FUNCTION_BLOCK "G269M_Code"
TITLE =G269M TEMPERATURE MES. KILN 1
//COPYRIGHT:    (C) 2009  BUHLER AG, CH-9240 UZWIL, SWITZERLAND
//
//PRODUCT:      WinCoS_BIW01_09
//
//TITLE:        TEMPERATURE MES. KILN 1
//                Machine group control
//                Maschinengruppensteuerung
//
//--------------------------------------------------------------------------------
//
//IDENT:        AUTHOR:             DEPT:                              DATE:
//
//P01_FB369.1.0 K.Renz              CSB41                              30.Sep.2009
//             1st Release
//
//--------------------------------------------------------------------------------
//
//PURPOSE:
//
//MANUAL :
//
//RESTRICTIONS:
//
//--------------------------------------------------------------------------------
AUTHOR : KR
FAMILY : USW
VERSION : 9.9


VAR
  Gr : "GCS7_GrpCtrlSub";	//Standard interface to group
  InOutValue1 : DINT ;	//Data for user
  InOutValue2 : DINT ;	//Data for user
  OutWayConflict : BOOL ;	//Data for user
  OutSelectionOk : BOOL ;	//Data for user
  CmdNewValue : BOOL ;	//Data for user
  CmdNewJob : BOOL ;	//Data for user
  OutCodeOK : BOOL ;	//Data for user
  InEndOfJob : BOOL ;	//Data for user
  staWayOk : BOOL ;	//Data for user
  EdgeStartRelease : BOOL ;	//Data for user
  read_3191 : BOOL ;	//Data for user
  USW9 : BOOL ;	//Data for user
  USW10 : BOOL ;	//Data for user
  USW11 : BOOL ;	//Data for user
  USW12 : BOOL ;	//Data for user
  USW13 : BOOL ;	//Data for user
  USW14 : BOOL ;	//Data for user
  USW15 : BOOL ;	//Data for user
  A_3191_BTE01 : "GCS7_E_AnalogInput";	// AnaInp
  A_3191_BTE05 : "GCS7_E_AnalogInput";	// AnaInp
  A_3191_BTE07 : "GCS7_E_AnalogInput";	// AnaInp
  A_3191_BTE08 : "GCS7_E_AnalogInput";	// AnaInp
  A_3191_BTE10 : "GCS7_E_AnalogInput";	// AnaInp
  A_3191_BTE11 : "GCS7_E_AnalogInput";	// AnaInp
  A_3191_BTE12 : "GCS7_E_AnalogInput";	// AnaInp
  A_3191_BTE06 : "GCS7_E_AnalogInput";	// AnaInp
  A_3191_BTE13 : "GCS7_E_AnalogInput";	// AnaInp
END_VAR
VAR_TEMP
  tmpEnable : BOOL ;
  tmpFlag : BOOL ;
  tmpCmdNext : BOOL ;
  tmpLocal : BOOL ;
  tmpAspOk : BOOL ;
  tmpHWStop : BOOL ;
  tmpInstanzDBNo : INT ;
END_VAR
BEGIN
NETWORK
TITLE =



NETWORK
TITLE =Read command from group control
//Parameter
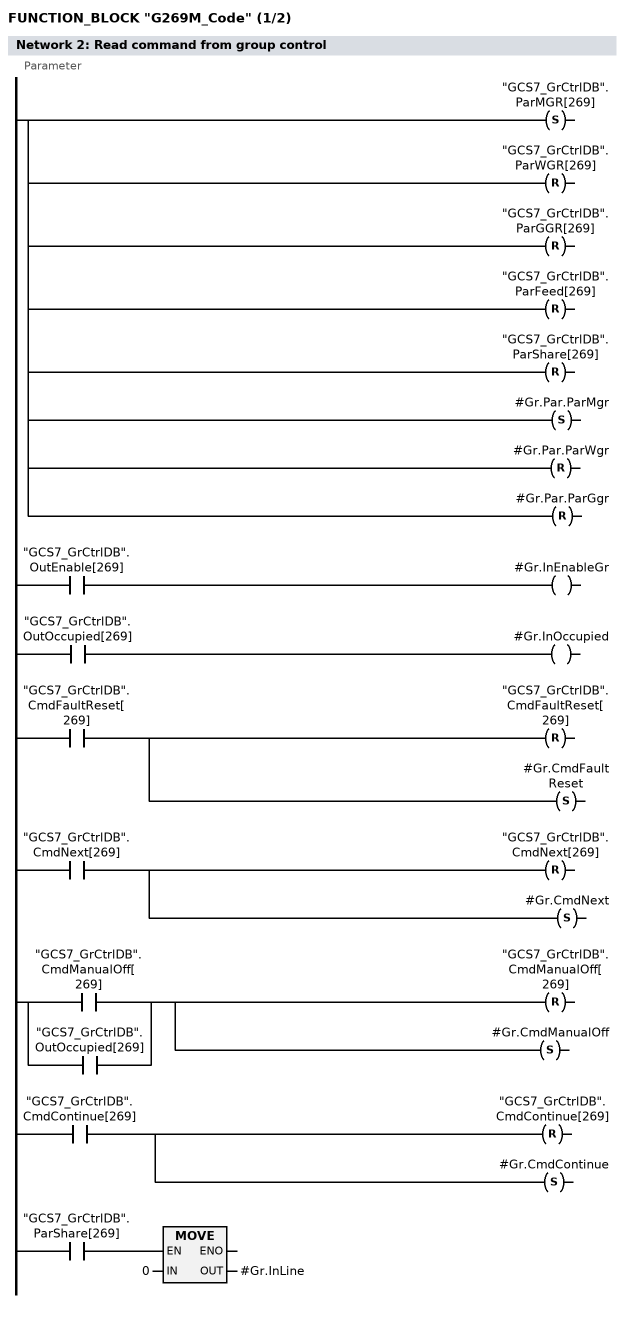
      SET   ;
      S     "GCS7_GrCtrlDB".ParMGR[269];
      R     "GCS7_GrCtrlDB".ParWGR[269];
      R     "GCS7_GrCtrlDB".ParGGR[269];
      R     "GCS7_GrCtrlDB".ParFeed[269];
      R     "GCS7_GrCtrlDB".ParShare[269];
      S     #Gr.Par.ParMgr;
      R     #Gr.Par.ParWgr;
      R     #Gr.Par.ParGgr;
//Command
      A     "GCS7_GrCtrlDB".OutEnable[269];
      =     #Gr.InEnableGr;
      A     "GCS7_GrCtrlDB".OutOccupied[269];
      =     #Gr.InOccupied;
      A     "GCS7_GrCtrlDB".CmdFaultReset[269];
      R     "GCS7_GrCtrlDB".CmdFaultReset[269];
      S     #Gr.CmdFaultReset;
      A     "GCS7_GrCtrlDB".CmdNext[269];
      R     "GCS7_GrCtrlDB".CmdNext[269];
      S     #Gr.CmdNext;
      A     "GCS7_GrCtrlDB".CmdManualOff[269];
      O     "GCS7_GrCtrlDB".OutOccupied[269];
      R     "GCS7_GrCtrlDB".CmdManualOff[269];
      S     #Gr.CmdManualOff;
      A     "GCS7_GrCtrlDB".CmdContinue[269];
      R     "GCS7_GrCtrlDB".CmdContinue[269];
      S     #Gr.CmdContinue;
//Init Line Number
      A     "GCS7_GrCtrlDB".ParShare[269];
      JCN   WE00;
      L     0;
      T     #Gr.InLine;
WE00: NOP   0;
NETWORK
TITLE =Call Methode Control
// 1. Handle Interface PCControl
// 2. Prepare mode --> ModePassive,ModeActive,ModeIdling
// 3. Reset global flags of the group
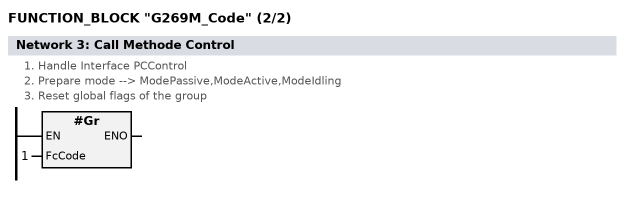
      CALL #Gr (
           FcCode                   := 1);
NETWORK
TITLE =Restart Idling Time

      L     #Gr.Par.ParIdling;
      L     2;
      >=I   ;
      JC    IdTm;
      T     #Gr.Par.ParIdling;
IdTm: NOP   0;
      CLR   ;
      S     #Gr.CmdRestartIdling;
NETWORK
TITLE =Prepare global flags



NETWORK
TITLE =Set Pattern (Target position)



NETWORK
TITLE =Interlocking WayOk



NETWORK
TITLE =Interlocking Autostart

      CLR   ;
      R     #Gr.OutAutostart;
NETWORK
TITLE =Interlocking Enable
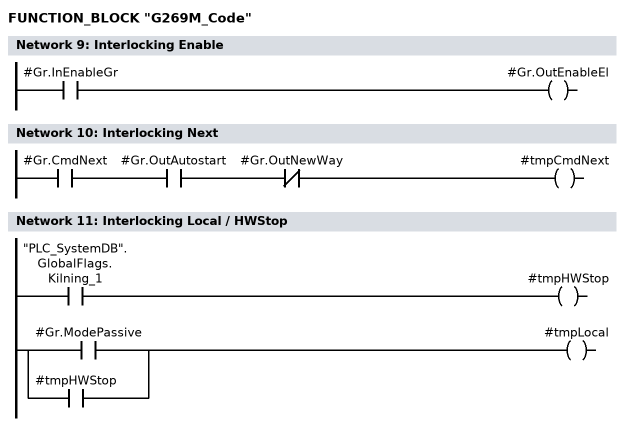

      A     #Gr.InEnableGr;
      =     #Gr.OutEnableEl;

NETWORK
TITLE =Interlocking Next

      A     #Gr.CmdNext;
      A     #Gr.OutAutostart;
      AN    #Gr.OutNewWay;
      =     #tmpCmdNext;

NETWORK
TITLE =Interlocking Local / HWStop

      A     "PLC_SystemDB".GlobalFlags.Kilning_1;
      =     #tmpHWStop;

      A     #Gr.ModePassive;
      O     #tmpHWStop;
      =     #tmpLocal;

NETWORK
TITLE ==A-3191-BTE01 : AIR TEMPERATURE BELOW FLOOR

      NOP   0;
//-InLocal---
      A     #tmpLocal;
      =     #A_3191_BTE01.InLocal;
//
//-Monitoring---
      A     "MAL1S032Par".Par.FlagProcess.ProcessActive;
      =     #A_3191_BTE01.InMonLL;
      =     #A_3191_BTE01.InMonL;
      CLR   ;
      =     #A_3191_BTE01.InMonMid;
      A     "MAL1S032Par".Par.FlagProcess.ProcessActive;
      =     #A_3191_BTE01.InMonH;
      =     #A_3191_BTE01.InMonHH;
//MW 2010.04.08
      SET   ;
      =     #A_3191_BTE01.Par.ParWarningL;
      =     #A_3191_BTE01.Par.ParWarningH;
      CLR   ;
      =     #A_3191_BTE01.Par.ParWarningLL;
      =     #A_3191_BTE01.Par.ParPreAlarmLL;
      =     #A_3191_BTE01.Par.ParPreAlarmHH;
      =     #A_3191_BTE01.Par.ParWarningHH;
//
//-Read inputs---
      L     "A_3191_BTE01_AI1";
      L     50;
      -I    ;
      T     #A_3191_BTE01.InpValue;
      A     "PLC_SystemDB".GlobalFlags.Kilning_1;
      =     #A_3191_BTE01.InHWStop;
      A     "PLC_DPInfo".Master[1].SlavesError[92];
      =     #A_3191_BTE01.InDPFault;
//
//-Set Parameters---
      SET   ; //BRT20100828 - kein Alarmhorn wenn Warning
      =     "G269M".A_3191_BTE01.Par.ParNoHornByWarning;

      AN    "MAL1S032Par".Par.FlagProcess.ProcessActive;
      JC    fui;
// Toleranzband -1,5°C Temperatur unter der Horde
      L     "MAL1S032Par".StepAct.TemperaturBelowFloor;
      L     L#10;
      *D    ;
      L     L#150; // =1,5°C
      -D    ;
      T     #A_3191_BTE01.Par.ParLimitL;
// Toleranzband +1,5°C Temperatur unter der Horde
      L     "MAL1S032Par".StepAct.TemperaturBelowFloor;
      L     L#10;
      *D    ;
      L     L#150; // =1,5°C
      +D    ;
      T     #A_3191_BTE01.Par.ParLimitH;
      JU    hui;
fui:  NOP   0;
      L     L#-10000; // -100,00°C
      T     #A_3191_BTE01.Par.ParLimitLL;
      L     L#0; // 0,00°C
      T     #A_3191_BTE01.Par.ParLimitL;
      L     L#9900; // 99,00°C
      T     #A_3191_BTE01.Par.ParLimitH;
      L     L#10000; // 100,00°C
      T     #A_3191_BTE01.Par.ParLimitHH;
hui:  NOP   0;
//
//-Call object control---
      CALL #A_3191_BTE01 ;
//
//-Write outputs---
// Schaltpunkt zu Oeffnen der Defrosterklappe
      L     #A_3191_BTE01.OutValuePc;
      L     7000; // =70,00°C
      >=I   ;
      =     "MAL1S032Par".Par.FlagProcess2.Schaltp_70;

NETWORK
TITLE ==A-3191-BTE05 : AIR TEMPERATURE DIFFUSOR FAN 1

      NOP   0;
//-InLocal---
      A     #tmpLocal;
      =     #A_3191_BTE05.InLocal;
//
//-Monitoring---
      CLR   ;
      =     #A_3191_BTE05.InMonLL;
      CLR   ;
      =     #A_3191_BTE05.InMonL;
      CLR   ;
      =     #A_3191_BTE05.InMonMid;
      CLR   ;
      =     #A_3191_BTE05.InMonH;
      A     "MAL1S032Par".Par.FlagProcess.ProcessActive;
      =     #A_3191_BTE05.InMonHH;
//
//-Read inputs---
      L     "A_3191_BTE05_AI1";
      L     50;
      -I    ;
      T     #A_3191_BTE05.InpValue;
      A     "PLC_SystemDB".GlobalFlags.Kilning_1;
      =     #A_3191_BTE05.InHWStop;
      A     "PLC_DPInfo".Master[1].SlavesError[92];
      =     #A_3191_BTE05.InDPFault;
//
//-Set Parameters---
      A     "MAL1S032Par".Par.FlagProcess.ProcessActive;
      R     #A_3191_BTE05.Par.ParNoHornByWarning;

      AN    "MAL1S032Par".Par.FlagProcess.ProcessActive;
      ON    "G271M".A_3125_MXZ01MA.Ma.StStartedFwd;
      ON    "G276M".A_3161_KCL12_REG_ON.StTrue;
      JC    fui1;

// Toleranzband -3,5°C Temperatur unter der Horde
      L     "MAL1S032Par".StepAct.TemperaturBelowFloor;
      L     L#10;
      *D    ;
      L     L#350; // =3,5°C
      -D    ;
      T     #A_3191_BTE05.Par.ParLimitL;
// Toleranzband +3,5°C Temperatur unter der Horde
      L     "MAL1S032Par".StepAct.TemperaturBelowFloor;
      L     L#10;
      *D    ;
      L     L#350; // =3,5°C
      +D    ;
      T     #A_3191_BTE05.Par.ParLimitH;
      JU    hui1;
fui1: NOP   0;


      L     L#-10000; // -100,00°C
      T     #A_3191_BTE05.Par.ParLimitLL;
      L     L#0; // 0,00°C
      T     #A_3191_BTE05.Par.ParLimitL;
      L     L#9900; // 99,00°C
      T     #A_3191_BTE05.Par.ParLimitH;
      L     L#10000; // 100,00°C
      T     #A_3191_BTE05.Par.ParLimitHH;
hui1: NOP   0;
//
//-Call object control---
      CALL #A_3191_BTE05 ;
//
//-Write outputs---
NETWORK
TITLE ==A-3191-BTE07 : AIR TEMPERATURE ABOVE FLOOR

      NOP   0;
//-InLocal---
      A     #tmpLocal;
      =     #A_3191_BTE07.InLocal;
//
//-Monitoring---
      CLR   ;
      =     #A_3191_BTE07.InMonLL;
      CLR   ;
      =     #A_3191_BTE07.InMonL;
      CLR   ;
      =     #A_3191_BTE07.InMonMid;
      A     "MAL1S032Par".Par.FlagProcess.ProcessActive;
      =     #A_3191_BTE07.InMonH;
      A     "MAL1S032Par".Par.FlagProcess.ProcessActive;
      AN    #A_3191_BTE07.OutOverflow;
      =     #A_3191_BTE07.Par.ParWarningH;
      A     "MAL1S032Par".Par.FlagProcess.ProcessActive;
      =     #A_3191_BTE07.InMonHH;
      =     #A_3191_BTE07.Par.ParPreAlarmHH;
      A     "MAL1S032Par".Par.FlagProcess.ProcessActive;
      AN    #A_3191_BTE07.OutOverflow;
      =     #A_3191_BTE07.Par.ParWarningHH;
//
//-Read inputs---
      L     "A_3191_BTE07_AI1";
      T     #A_3191_BTE07.InpValue;
      A     "PLC_SystemDB".GlobalFlags.Kilning_1;
      =     #A_3191_BTE07.InHWStop;
      A     "PLC_DPInfo".Master[1].SlavesError[92];
      =     #A_3191_BTE07.InDPFault;
//
//-Set Parameters---
      A     "MAL1S032Par".Par.FlagProcess.ProcessActive;
      R     #A_3191_BTE07.Par.ParNoHornByWarning;

      AN    "MAL1S032Par".Par.FlagProcess.ProcessActive;
      JC    psp;
//      L     "MAL1S032Par".RecipeHeader.WarningTempAboveFloor
      L     L#900; // 90,00°C
      L     L#10;
      *D    ;
      T     #A_3191_BTE07.Par.ParLimitH;
      L     #A_3191_BTE07.Par.ParLimitH;
      L     L#500;
      +D    ;
      T     #A_3191_BTE07.Par.ParLimitHH;
psp:  NOP   0;
      A     "MAL1S032Par".Par.FlagProcess.ProcessActive;
      JC    npsp;
      L     L#-10000; // -100,00°C
      T     #A_3191_BTE07.Par.ParLimitLL;
      L     L#0; // 0,00°C
      T     #A_3191_BTE07.Par.ParLimitL;
      L     L#9900; // 99,00°C
      T     #A_3191_BTE07.Par.ParLimitH;
      L     L#10000; // 100,00°C
      T     #A_3191_BTE07.Par.ParLimitHH;
npsp: NOP   0;
//
//-Call object control---
      CALL #A_3191_BTE07 ;
//
//-Write outputs---
NETWORK
TITLE ==A-3191-BTE08 : AIR TEMPERATURE AFTER BURNER 1
//      NOP   0
////-InLocal---
//      U     #tmpLocal
//      =     #A_3191_BTE08.InLocal
//
////-Monitoring---
//      CLR
//      =     #A_3191_BTE08.InMonLL
//      CLR
//      =     #A_3191_BTE08.InMonL
//      CLR
//      =     #A_3191_BTE08.InMonMid
//      CLR
//      =     #A_3191_BTE08.InMonH
//      U     "MAL1S032Par".Par.FlagProcess.ProcessActive
//      =     #A_3191_BTE08.InMonHH
////
////-Read inputs---
//      L     "A_3191_BTE08_AI1"
//      T     #A_3191_BTE08.InpValue
//      U     "PLC_SystemDB".GlobalFlags.Kilning_1
//      =     #A_3191_BTE08.InHWStop
//      U     "PLC_DPInfo".Master[1].SlavesError[92]
//      =     #A_3191_BTE08.InDPFault
////
////-Set Parameters---
//      L     L#-10000                    // -100,00°C
//      T     #A_3191_BTE08.Par.ParLimitLL
//      L     L#0                         // 0,00°C
//      T     #A_3191_BTE08.Par.ParLimitL
//      L     L#9900                      // 99,00°C
//      T     #A_3191_BTE08.Par.ParLimitH
//      L     L#10000                     // 100,00°C
//      T     #A_3191_BTE08.Par.ParLimitHH
////
////-Call object control---
//      CALL  #A_3191_BTE08
////
////-Write outputs---
//


NETWORK
TITLE ==A-3191-BTE10 : AIR TEMPERATURE BEFORE BURNER 2

      NOP   0;
//-InLocal---
      A     #tmpLocal;
      =     #A_3191_BTE10.InLocal;
//
//-Monitoring---
      CLR   ;
      =     #A_3191_BTE10.InMonLL;
      CLR   ;
      =     #A_3191_BTE10.InMonL;
      CLR   ;
      =     #A_3191_BTE10.InMonMid;
      CLR   ;
      =     #A_3191_BTE10.InMonH;
      A     "MAL1S032Par".Par.FlagProcess.ProcessActive;
      =     #A_3191_BTE10.InMonHH;
//
//-Read inputs---
      L     "A_3191_BTE10_AI1";
      T     #A_3191_BTE10.InpValue;
      A     "PLC_SystemDB".GlobalFlags.Kilning_1;
      =     #A_3191_BTE10.InHWStop;
      A     "PLC_DPInfo".Master[1].SlavesError[92];
      =     #A_3191_BTE10.InDPFault;
//
//-Set Parameters---
      L     L#-10000; // -100,00°C
      T     #A_3191_BTE10.Par.ParLimitLL;
      L     L#0; // 0,00°C
      T     #A_3191_BTE10.Par.ParLimitL;
      L     L#9900; // 99,00°C
      T     #A_3191_BTE10.Par.ParLimitH;
      L     L#10000; // 100,00°C
      T     #A_3191_BTE10.Par.ParLimitHH;
//
//-Call object control---
      CALL #A_3191_BTE10 ;
//
//-Write outputs---
NETWORK
TITLE ==A-3191-BTE11 : AIR TEMPERATURE AMBIENT AIR

      NOP   0;
//-InLocal---
      A     #tmpLocal;
      =     #A_3191_BTE11.InLocal;
//
//-Monitoring---
      SET   ;
      =     #A_3191_BTE11.InMonLL;
      CLR   ;
      =     #A_3191_BTE11.InMonL;
      CLR   ;
      =     #A_3191_BTE11.InMonMid;
      CLR   ;
      =     #A_3191_BTE11.InMonH;
      SET   ;
      =     #A_3191_BTE11.InMonHH;
//
//-Read inputs---
      L     "A_3191_BTE11_AI1";
      T     #A_3191_BTE11.InpValue;
      A     "PLC_SystemDB".GlobalFlags.Kilning_1;
      =     #A_3191_BTE11.InHWStop;
      A     "PLC_DPInfo".Master[1].SlavesError[92];
      =     #A_3191_BTE11.InDPFault;
//
//-Set Parameters---
      A     "MAL1S032Par".Par.FlagProcess.ProcessActive;
      R     #A_3191_BTE11.Par.ParNoHornByWarning;

      L     L#-10000; // -100,00°C
      T     #A_3191_BTE11.Par.ParLimitLL;
      L     L#0; // 0,00°C
      T     #A_3191_BTE11.Par.ParLimitL;
      L     L#3200; // 32,00°C
//      L     "MAL1Par".Values1.Value03   // Line Parameter --> not used!!
//      L     L#100
//      *D
      T     #A_3191_BTE11.Par.ParLimitH;
      L     L#10000; // 100,00°C
      T     #A_3191_BTE11.Par.ParLimitHH;
//
//-Call object control---
      CALL #A_3191_BTE11 ;
//
//-Write outputs---
NETWORK
TITLE ==A-3191-BTE13 : AIR TEMPERATURE BEFORE HEAT EXCHANGER
//invented by Butrim to monitor exchanger EFFICIENCY FACTOR lol
      NOP   0;
//-InLocal---
      A     #tmpLocal;
      =     #A_3191_BTE13.InLocal;

//-Monitoring---
      SET   ;
      =     #A_3191_BTE13.InMonLL;
      CLR   ;
      =     #A_3191_BTE13.InMonL;
      CLR   ;
      =     #A_3191_BTE13.InMonMid;
      CLR   ;
      =     #A_3191_BTE13.InMonH;
      SET   ;
      =     #A_3191_BTE13.InMonHH;
//
//-Read inputs---
//L     "A_3191_BTE11_AI1"
      L     PIW 1046;
      T     #A_3191_BTE13.InpValue;
      A     "PLC_SystemDB".GlobalFlags.Kilning_1;
      =     #A_3191_BTE13.InHWStop;
      A     "PLC_DPInfo".Master[1].SlavesError[92];
      =     #A_3191_BTE13.InDPFault;
//
//-Set Parameters---
      A     "MAL1S032Par".Par.FlagProcess.ProcessActive;
      R     #A_3191_BTE13.Par.ParNoHornByWarning;

      L     L#-10000; // -100,00°C
      T     #A_3191_BTE13.Par.ParLimitLL;
      L     L#0; // 0,00°C
      T     #A_3191_BTE13.Par.ParLimitL;
      L     L#9900; // 99,00°C
      T     #A_3191_BTE13.Par.ParLimitH;
      L     L#10000; // 100,00°C
      T     #A_3191_BTE13.Par.ParLimitHH;
//
//-Call object control---
      CALL #A_3191_BTE13 ;
//
//-Write outputs---


NETWORK
TITLE ==A-3191-BTE12 : AIR TEMPERATURE AFTER HEAT EXCHANGER FLAP

      NOP   0;
//-InLocal---
      A     #tmpLocal;
      =     #A_3191_BTE12.InLocal;
//
//-Monitoring---
      CLR   ;
      =     #A_3191_BTE12.InMonLL;
      CLR   ;
      =     #A_3191_BTE12.InMonL;
      CLR   ;
      =     #A_3191_BTE12.InMonMid;
      CLR   ;
      =     #A_3191_BTE12.InMonH;
      A     "MAL1S032Par".Par.FlagProcess.ProcessActive;
      =     #A_3191_BTE12.InMonHH;
//
//-Read inputs---
      L     "A_3191_BTE12_AI1";
      T     #A_3191_BTE12.InpValue;
      A     "PLC_SystemDB".GlobalFlags.Kilning_1;
      =     #A_3191_BTE12.InHWStop;
      A     "PLC_DPInfo".Master[1].SlavesError[92];
      =     #A_3191_BTE12.InDPFault;
//
//-Set Parameters---
      L     L#-10000; // -100,00°C
      T     #A_3191_BTE12.Par.ParLimitLL;
      L     L#0; // 0,00°C
      T     #A_3191_BTE12.Par.ParLimitL;
      L     L#9900; // 99,00°C
      T     #A_3191_BTE12.Par.ParLimitH;
      L     L#10000; // 100,00°C
      T     #A_3191_BTE12.Par.ParLimitHH;
//
//-Call object control---
      CALL #A_3191_BTE12 ;
//
//-Write outputs---
NETWORK
TITLE ==A-3191-BTE06 : AIR TEMPERATURE DIFFUSOR FAN 2

      NOP   0;
//-InLocal---
      A     #tmpLocal;
      =     #A_3191_BTE06.InLocal;
//
//-Monitoring---
      CLR   ;
      =     #A_3191_BTE06.InMonLL;
      CLR   ;
      =     #A_3191_BTE06.InMonL;
      CLR   ;
      =     #A_3191_BTE06.InMonMid;
      CLR   ;
      =     #A_3191_BTE06.InMonH;
      A     "MAL1S032Par".Par.FlagProcess.ProcessActive;
      =     #A_3191_BTE06.InMonHH;
//
//-Read inputs---
      L     "A_3191_BTE06_AI1";
      L     50;
      -I    ;
      T     #A_3191_BTE06.InpValue;
      A     "PLC_SystemDB".GlobalFlags.Kilning_1;
      =     #A_3191_BTE06.InHWStop;
      A     "PLC_DPInfo".Master[1].SlavesError[92];
      =     #A_3191_BTE06.InDPFault;
//
//-Set Parameters---
      A     "MAL1S032Par".Par.FlagProcess.ProcessActive;
      R     #A_3191_BTE06.Par.ParNoHornByWarning;

      AN    "MAL1S032Par".Par.FlagProcess.ProcessActive;
      ON    "G271M".A_3126_MXZ01MA.Ma.StStartedFwd;
      ON    "G276M".A_3161_KCL12_REG_ON.StTrue;
      JC    fui2;

// Toleranzband -3,5°C Temperatur unter der Horde
      L     "MAL1S032Par".StepAct.TemperaturBelowFloor;
      L     L#10;
      *D    ;
      L     L#350; // =3,5°C
      -D    ;
      T     #A_3191_BTE06.Par.ParLimitL;
// Toleranzband +3,5°C Temperatur unter der Horde
      L     "MAL1S032Par".StepAct.TemperaturBelowFloor;
      L     L#10;
      *D    ;
      L     L#350; // =3,5°C
      +D    ;
      T     #A_3191_BTE06.Par.ParLimitH;
      JU    hui2;
fui2: NOP   0;

      L     L#-10000; // -100,00°C
      T     #A_3191_BTE06.Par.ParLimitLL;
      L     L#0; // 0,00°C
      T     #A_3191_BTE06.Par.ParLimitL;
      L     L#9900; // 99,00°C
      T     #A_3191_BTE06.Par.ParLimitH;
      L     L#10000; // 100,00°C
      T     #A_3191_BTE06.Par.ParLimitHH;
hui2: NOP   0;
//
//-Set Parameters---
//
//-Call object control---
      CALL #A_3191_BTE06 ;
//
//-Write outputs---
NETWORK
TITLE =Test Fault
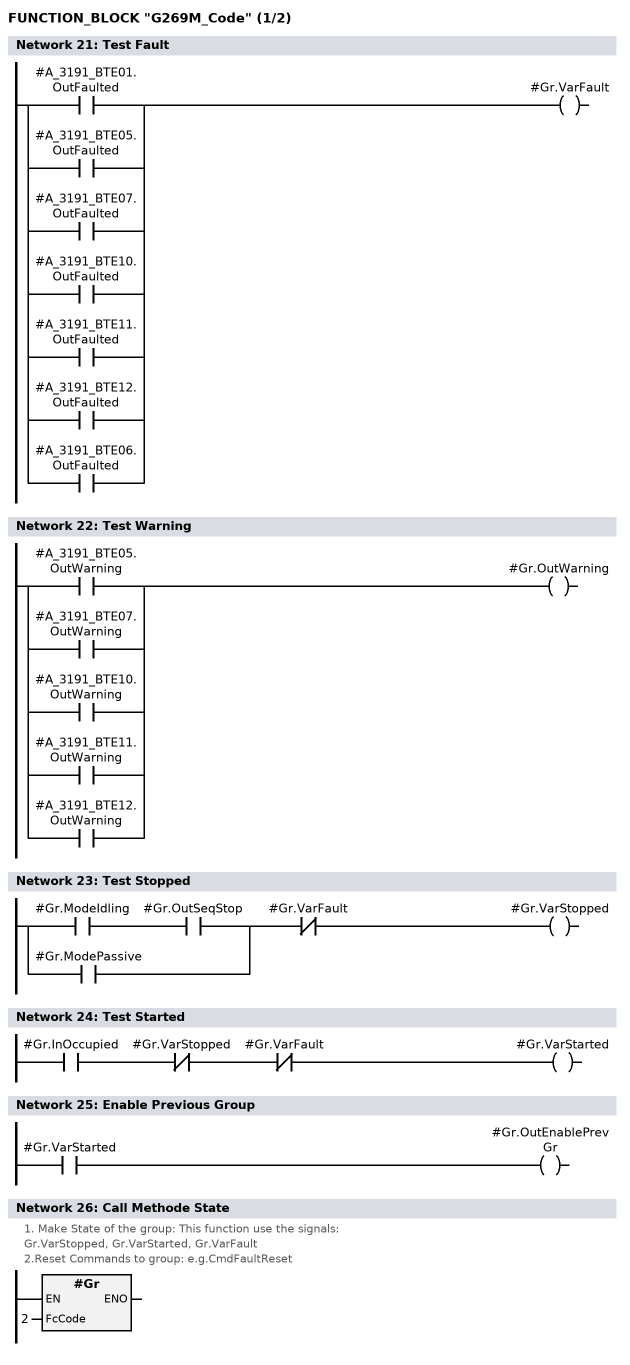

      A     #A_3191_BTE01.OutFaulted;
      O     #A_3191_BTE05.OutFaulted;
      O     #A_3191_BTE07.OutFaulted;
//      O     #A_3191_BTE08.OutFaulted
      O     #A_3191_BTE10.OutFaulted;
      O     #A_3191_BTE11.OutFaulted;
      O     #A_3191_BTE12.OutFaulted;
      O     #A_3191_BTE06.OutFaulted;
      =     #Gr.VarFault;
NETWORK
TITLE =Test Warning

//      U     #A_3191_BTE01.OutWarning
      O     #A_3191_BTE05.OutWarning;
      O     #A_3191_BTE07.OutWarning;
//      O     #A_3191_BTE08.OutWarning
      O     #A_3191_BTE10.OutWarning;
      O     #A_3191_BTE11.OutWarning;
      O     #A_3191_BTE12.OutWarning;
      =     #Gr.OutWarning;
NETWORK
TITLE =Test Stopped

      A     #Gr.ModeIdling;
      A     #Gr.OutSeqStop;
      O     #Gr.ModePassive;
      AN    #Gr.VarFault;
      =     #Gr.VarStopped;
NETWORK
TITLE =Test Started

      A     #Gr.InOccupied;
      AN    #Gr.VarStopped;
      AN    #Gr.VarFault;
      =     #Gr.VarStarted;
NETWORK
TITLE =Enable Previous Group

      A     #Gr.VarStarted;
      =     #Gr.OutEnablePrevGr;
NETWORK
TITLE =Call Methode State
//1. Make State of the group: This function use the signals:
//        Gr.VarStopped, Gr.VarStarted, Gr.VarFault
//2.Reset Commands to group: e.g.CmdFaultReset
      CALL #Gr (
           FcCode                   := 2);
NETWORK
TITLE =Init
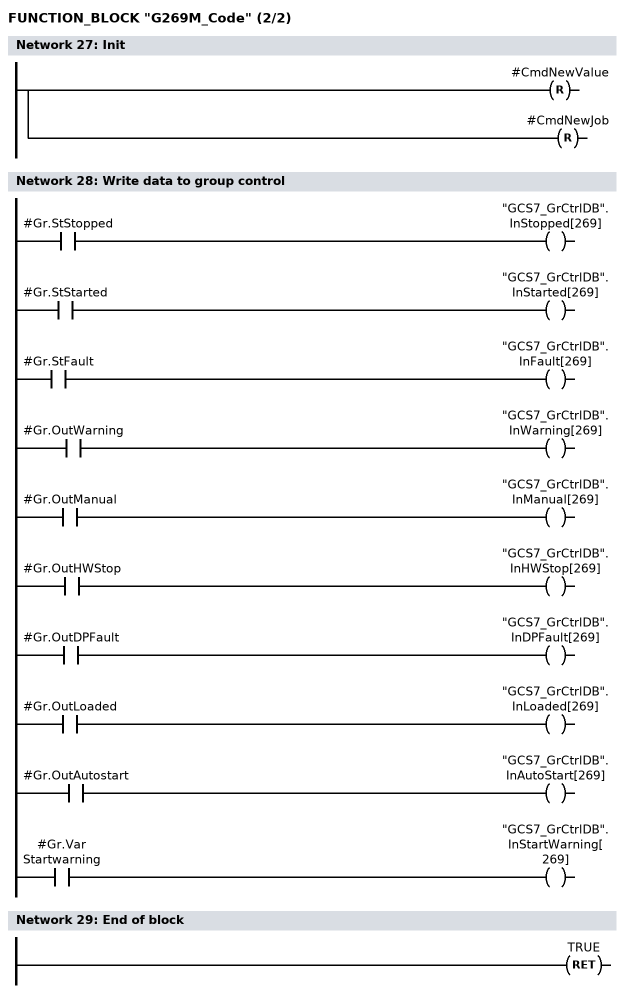

      SET   ;
      R     #CmdNewValue;
      R     #CmdNewJob;
NETWORK
TITLE =Write data to group control

      A     #Gr.StStopped;
      =     "GCS7_GrCtrlDB".InStopped[269];
      A     #Gr.StStarted;
      =     "GCS7_GrCtrlDB".InStarted[269];
      A     #Gr.StFault;
      =     "GCS7_GrCtrlDB".InFault[269];
      A     #Gr.OutWarning;
      =     "GCS7_GrCtrlDB".InWarning[269];
      A     #Gr.OutManual;
      =     "GCS7_GrCtrlDB".InManual[269];
      A     #Gr.OutHWStop;
      =     "GCS7_GrCtrlDB".InHWStop[269];
      A     #Gr.OutDPFault;
      =     "GCS7_GrCtrlDB".InDPFault[269];
      A     #Gr.OutLoaded;
      =     "GCS7_GrCtrlDB".InLoaded[269];
      A     #Gr.OutAutostart;
      =     "GCS7_GrCtrlDB".InAutoStart[269];
      A     #Gr.VarStartwarning;
      =     "GCS7_GrCtrlDB".InStartWarning[269];
NETWORK
TITLE =End of block

      BE    ;

END_FUNCTION_BLOCK

